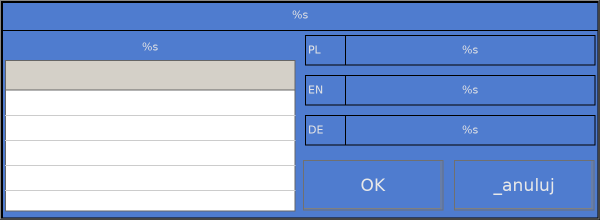
VISUALIZATION D_AddRecipe  // 600x220
VAR_IN_OUT
	{attribute "VAR_IN_OUT_AS_POINTER}
	stData		: ST_MCHMIPrepareScreen_02_XX_AddRecipe;
END_VAR
    Rectangle (0,0 600x220)
    Rectangle (305,35 290x30), "PL"
    Line (0,30) (600,30)
    Rectangle (3,3 594x24), "%s", text variable: stData.wsTitle
    Button (454,160 140x50), "_anuluj", text list: 'TextListGlobal', text index: 2
        OnMouseDown: execute { stData.bCancel := TRUE; }
        OnMouseUp: CloseDialog Dialog=D_AddRecipe, Result=Ignore, NumpadKeypadSet=True
    Button (303,160 140x50), "OK"
        OnMouseDown: execute { stData.bOk := TRUE; }
        OnMouseUp: CloseDialog Dialog=D_AddRecipe, Result=OK, NumpadKeypadSet=True
    Rectangle (345,35 250x30), "%s", text variable: stData.stNewNames.arrText [1]
        OnMouseDown: write the text variable via KlawiaturaLitery
    Rectangle (305,75 290x30), "EN"
    Rectangle (345,75 250x30), "%s", text variable: stData.stNewNames.arrText [2]
        OnMouseDown: write the text variable via KlawiaturaLitery
    Rectangle (305,115 290x30), "DE"
    Rectangle (345,115 250x30), "%s", text variable: stData.stNewNames.arrText [3]
        OnMouseDown: write the text variable via KlawiaturaLitery
    Rectangle (3,35 294x24), "%s", text variable: stData.wsSource
    Table (5,60 290x151), data array: stData.arrListOfName
        p3854506369: stData.arrListOfName[INDEX]
        p1128707560: stData.iNumberOfNames
        p1822360349: stData.bSelectedRow
        p1137915858: stData.iSelectedName
END_VISUALIZATION

(* stored: Version 1.1.0.1
   Visu D_AddRecipe: Id {fb6b878c-b0ad-0d9c-24e4-93cbe8625aa5} *)
